# EPICS SNL sequencer program: siteApps/SRF-HWR-Cooldown-1-0/srfcooldownApp/src/sncSRFCooldown.stt
program sncSRFCooldown
option +r;

%%#include <math.h>

char SRF_HWRB01_Valve[40] = "SRF01-Bunker1:HWRB01-Valve";

char    valvename[60];
float   valveval;
assign  valveval to "";

string steppv;
assign steppv to "{SYS}{SUBSYS}{DEV}{SUBDEV}StepPV";
monitor steppv;

int ss_start = 0;
assign ss_start to "{SYS}{SUBSYS}{DEV}{SUBDEV}Start";
monitor ss_start;
evflag	efStop;
sync ss_start to efStop;

int		phaseend;
assign	phaseend to "{SYS}{SUBSYS}{DEV}{SUBDEV}PhaseEnd";
monitor phaseend;

float cdDelay;
assign cdDelay to "{SYS}{SUBSYS}{DEV}{SUBDEV}StepDly";
monitor cdDelay;

//Valve Control
char    logicname[60];
int     proc = 1;
assign  proc to "";

ss ssSRFCooldown
{
	state Init
	{
		when(TRUE)
		{
			printf("Wait Cooldown Logic Process!!\n");
			strcpy(steppv, "Wait Cooldown Proc");
			pvPut(steppv, SYNC);
		}state Stop
	}
    state Stop
    {
        when(ss_start == 1)
        {
			sprintf(logicname,   "%s:CDLogic.PROC", SRF_HWRB01_Valve);
			pvAssign(proc, logicname);
			pvMonitor(proc);

			sprintf(valvename,   "%s:CDLogic.L",    SRF_HWRB01_Valve);
			pvAssign(valveval, valvename);
			pvMonitor(valveval);

			printf("Started Cooldown!!\n");
			strcpy(steppv, "Started Cooldown");
			pvPut(steppv, SYNC);

        }state SRFCooldown
    }

	state SRFCooldown
	{
		when(delay(cdDelay) && phaseend < 1 && ss_start == 1)
		{
			proc = 1;
			pvPut(proc, SYNC);

			printf("Processing Cooldown Logic !!\n");
			strcpy(steppv, "Processing Cooldown");
			pvPut(steppv, SYNC);
		}state SRFCooldown

		when(delay(cdDelay) && phaseend >= 1  && ss_start != 1 )
		{
			pvStopMonitor(valveval);
			pvStopMonitor(proc);

			strcpy(steppv, "Stopped Cooldown");
			pvPut(steppv, SYNC);
		}state PhaseEnd
	}

	state PhaseEnd
	{
		when(delay(cdDelay) && ss_start != 1)
		{
			ss_start = 0;
			pvPut(ss_start, SYNC);

			strcpy(steppv, "Complete PhaseEnd");
			pvPut(steppv, SYNC);
		}state Stop
	}
}
